FUNCTION_BLOCK SUBSCRIBE_5 (* Subscribe to a PUBLISH_5 Block *)
  (* Description: Copyright (c) 2017 fortiss GmbH This program and the accompanying materials are made available under the terms of the Eclipse Public License 2.0 which is available at https://www.eclipse.org/legal/epl-2.0/ SPDX-License-Identifier: EPL-2.0 *)
  (* Version 3.0, 2025-04-14, Patrick Aigner, changed package *)
  (* Version 1.0, 2017-10-25, Alois Zoitl, fortiss GmbH, initial API and implementation and/or initial documentation *)
  PACKAGE iec61499::net;
  {SET_ATTRIBUTE(eclipse4diac::core::GenericClassName, 'GEN_SUBSCRIBE')}
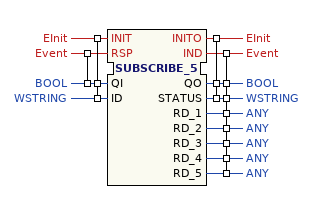
  EVENT_INPUT
    INIT : EInit WITH QI, ID; (* Initialization *)
    RSP WITH QI;
  END_EVENT
  EVENT_OUTPUT
    INITO : EInit WITH QO, STATUS; (* Initialization Confirm *)
    IND WITH QO, STATUS, RD_1, RD_3, RD_2, RD_4, RD_5; (* New data available *)
  END_EVENT
  VAR_INPUT
    QI : BOOL;
    ID : WSTRING;
  END_VAR
  VAR_OUTPUT
    QO : BOOL;
    STATUS : WSTRING;
    RD_1 : ANY;
    RD_2 : ANY;
    RD_3 : ANY;
    RD_4 : ANY;
    RD_5 : ANY;
  END_VAR
END_FUNCTION_BLOCK
